// Mitsubishi GX Works2 project: 20240318_AI机程序新增MODBUS-通道1   PLC: FX3S

PROGRAM MAIN
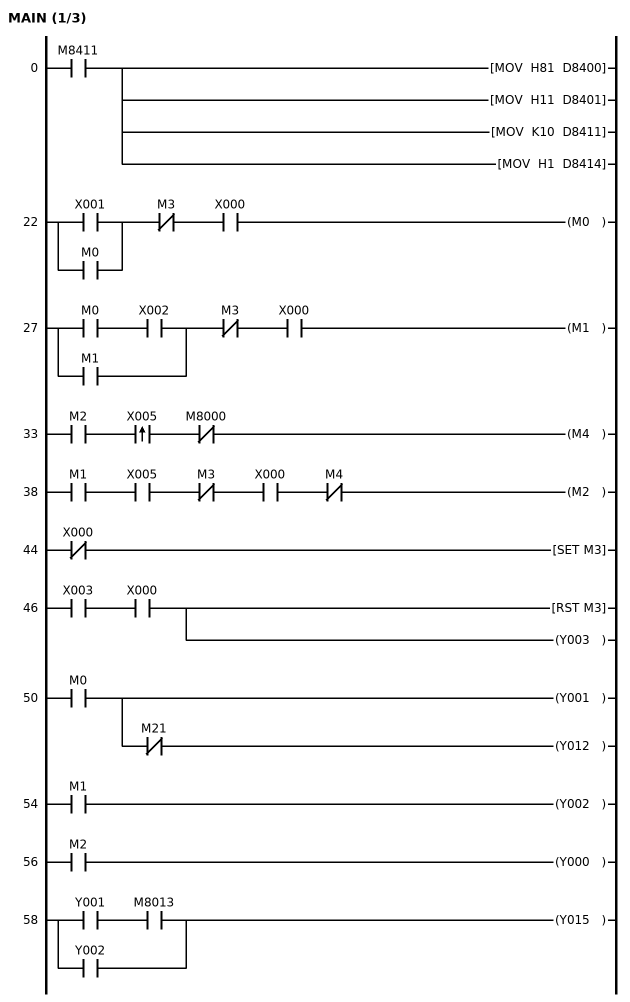
0     LD      M8411
      MOV     H81 D8400
      MOV     H11 D8401
      MOV     K10 D8411
      MOV     H1 D8414
22    LD      X001
      OR      M0
      ANI     M3
      AND     X000
      OUT     M0
27    LD      M0
      AND     X002
      OR      M1
      ANI     M3
      AND     X000
      OUT     M1
33    LD      M2
      ANDP    X005
      ANI     M8000
      OUT     M4
38    LD      M1
      AND     X005
      ANI     M3
      AND     X000
      ANI     M4
      OUT     M2
44    LDI     X000
      SET     M3
46    LD      X003
      AND     X000
      RST     M3
      OUT     Y003
50    LD      M0
      OUT     Y001
      ANI     M21
      OUT     Y012
54    LD      M1
      OUT     Y002
56    LD      M2
      OUT     Y000
58    LD      Y001
      AND     M8013
      OR      Y002
      OUT     Y015
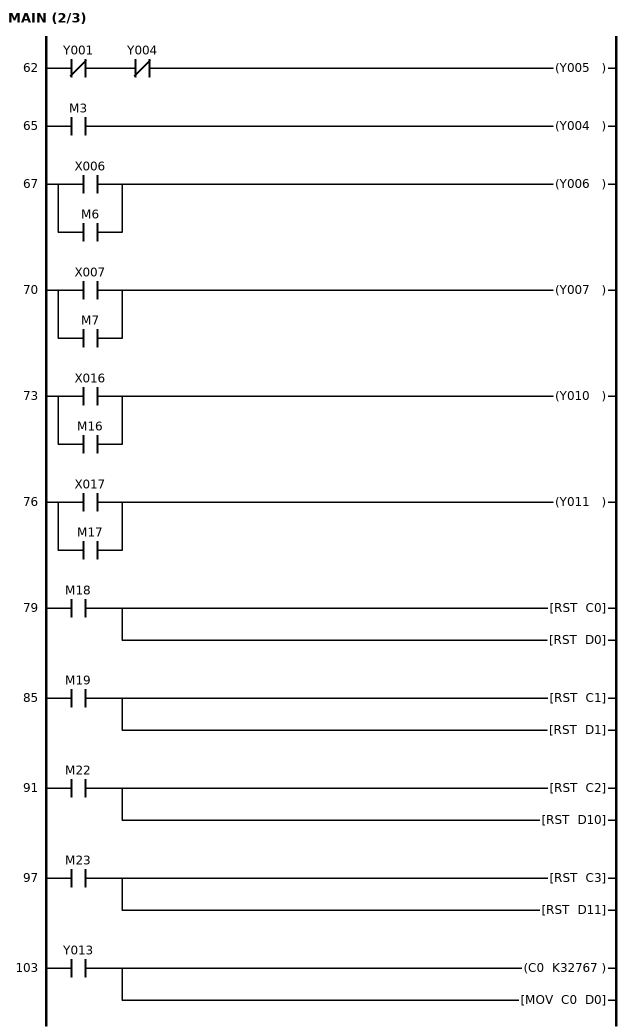
62    LDI     Y001
      ANI     Y004
      OUT     Y005
65    LD      M3
      OUT     Y004
67    LD      X006
      OR      M6
      OUT     Y006
70    LD      X007
      OR      M7
      OUT     Y007
73    LD      X016
      OR      M16
      OUT     Y010
76    LD      X017
      OR      M17
      OUT     Y011
79    LD      M18
      RST     C0
      RST     D0
85    LD      M19
      RST     C1
      RST     D1
91    LD      M22
      RST     C2
      RST     D10
97    LD      M23
      RST     C3
      RST     D11
103   LD      Y013
      OUT     C0 K32767
      MOV     C0 D0
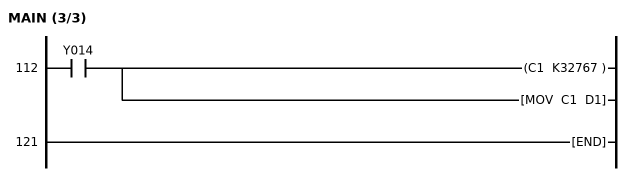
112   LD      Y014
      OUT     C1 K32767
      MOV     C1 D1
121   END
END_PROGRAM
